FUNCTION GetDefaultValue : string
VAR_INPUT
	DataType : STRING;
END_VAR
VAR
	defaultValue : STRING;
END_VAR

IF DataType = 'string' THEN
	defaultValue := '';
END_IF

GetDefaultValue := defaultValue;

END_FUNCTION

(* stored: Version 1.1.0.1, ProductVersion 3.1.4022.16
   POU GetDefaultValue: Id {1998dbda-6347-45ba-8a8e-8489af7dd1bd}, SpecialFunc None *)
